(* PLC project Proj_Ueb_sw01, Beckhoff Automation GmbH TwinCAT PLC Control 3.5.13.21 *)
(* stored: creationDateTime 2022-03-28T15:37:04.1596017, modificationDateTime 2022-03-28T15:37:04.1596017 *)

FUNCTION F_0to10V_TO_INT : INT
VAR_INPUT
	r_AnalogValue0to10V		: REAL;
END_VAR
VAR
	i_Val					: DINT;
END_VAR
VAR CONSTANT
	MAX_VOLTAGE				: REAL := 10.0;
	MAX_INT					: INT := 32767;
END_VAR

            // Multiply
i_Val := REAL_TO_DINT(r_AnalogValue0to10V * INT_TO_REAL(MAX_INT));

// divide by 10, convert to int
F_0to10V_TO_INT := DINT_TO_INT(i_Val / REAL_TO_INT(MAX_VOLTAGE));
          
END_FUNCTION
